TYPE (* IEC61131-3, Table 14#5 *)
  (* Standard: 1131-3 *)
  (* Version 0.0, 3/13/2026, Schneider Electric, Template *)
  PACKAGE Main;
  {SET_ATTRIBUTE(nxtDataType, yuBjJmbjdzTXbTqqCuFqqxQXJE5mK0LRrTxr6eXSk87W43s6zXXEgySxlizrayYEt1SYx1LTMSJ1NRBePvhs5dvgCqEZdX160HumpOPkI+BmhRDl9zNqgQ==)}
  Component_State : STRUCT
    name : STRING[150];
    state : INT;
  END_STRUCT;
END_TYPE
